// TIA Portal V19 export
DATA_BLOCK "ManualOperationControl_U2Em1"   // DB105
// stored: MemoryReserve 100
   VAR
      manualOperationEm { ExternalAccessible := 'False'; ExternalVisible := 'False'; ExternalWritable := 'False'} : "LAF_typeManEm";
      manualOperationEmArea { ExternalAccessible := 'False'; ExternalVisible := 'False'; ExternalWritable := 'False'} : Array[1..1] of "LAF_typeManOperationArea";
      manualOperationCms { ExternalAccessible := 'False'; ExternalVisible := 'False'; ExternalWritable := 'False'} : Array[1..1] of "LAF_typeManOperation";
   END_VAR
BEGIN
   manualOperationEm.equipmentModuleNum := 2010;
   manualOperationEmArea[1].displayedLines := '1';
END_DATA_BLOCK
